// Mitsubishi GX Works2 project: q7   PLC: Q02/Q02H

PROGRAM MAIN
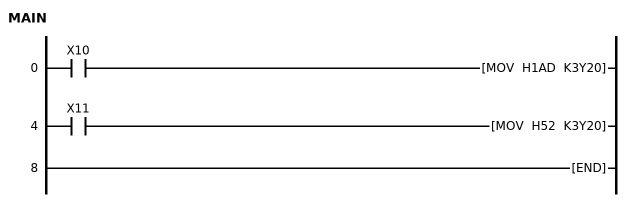
0     LD      X10
      MOV     H1AD K3Y20
4     LD      X11
      MOV     H52 K3Y20
8     END
END_PROGRAM
